FUNCTION xdotc_i : LREAL
VAR_INPUT
    b_n: DINT;
    x: ARRAY [0..24] OF LREAL;
    ix0: DINT;
    y: ARRAY [0..24] OF LREAL;
    iy0: DINT;
END_VAR
VAR
    ix: DINT;
    iy: DINT;
    k: DINT;
END_VAR

xdotc_i := 0.0;
IF b_n >= 1 THEN 
    ix := ix0;
    iy := iy0;
    k := 0;
    WHILE k <= (b_n - 1) DO
        xdotc_i := (x[ix - 1] * y[iy - 1]) + xdotc_i;
        ix := ix + 1;
        iy := iy + 1;
        k := k + 1;
    END_WHILE;
END_IF;

END_FUNCTION

(* stored: Version 1.1.0.1, ProductVersion 3.1.4024.12
   POU xdotc_i: Id {434704c9-6754-4b4f-8f47-61e4281c11de}, SpecialFunc None *)
